{attribute 'qualified_only'}
VAR_GLOBAL
	Remote_Panel_1:  Safety_Bypass_RemotePanel;
	Remote_Panel_2:  Safety_Bypass_RemotePanel;
END_VAR

(* stored: Version 1.1.0.1
   GVL Bypass: Id {3fa1d9fd-3a51-4976-b229-82ae4574f61f} *)
